Staubli VAL3: io_System.pjx

--- io_System.pjx ---
Parameters version=s7.0 stackSize=5000 millimeterUnit=true
Program file=_globals.pgx
Program file=InitSysIO.pgx
Program file=SysIN.pgx
Program file=SysOUT.pgx
Data file=io_System.dtx
Library alias=io path=Disk://io/io.pjx

--- io_System.dtx ---
public num nLiAuto
public num nLiAux1
public num nLiAux2
public num nLiAux3
public num nLiDoorOpen
public num nLiEnd
public num nLiHome = 1
public num nLiMouldFree
public num nLiPartMade
public num nLiRobotOff
public num nLiSafety
public num nLiStart
public num nLiStop = 1
public num nLiTotalHome = 1
public num nLiWarning
public num nStateRobot
public num nLiTowerRed
public num nLiTowerYellow
public num nLiTowerGreen
public num nPowerCountCtrl
public num nLastServiceCtr
public num nLastServiceArm
public num nServiceRemain
public string sAux1
public string sAux2
public bool bBlockedCycle
public bool bBlockedUser
public bool bBtEnd
public bool bBtHome
public bool bBtRobotOff
public bool bBtStart
public bool bBtStop
public bool bCancelHomeCycl
public bool bCycleEndCalled
public bool bCycleEndPos
public bool bEnd
public bool bF7
public bool bF8
public bool bF_End
public bool bF_Home
public bool bF_Off
public bool bF_Start
public bool bF_Stop
public bool bFirstRunAfterL = true
public bool bFlashFast
public bool bFlashSlow
public bool bForceHomeReq
public bool bForceHome_ = true
public bool bHomeRetActive
public bool bModified
public bool bMouldArmInPLC
public bool bPartMade
public bool bRobotHome = true
public bool bRobotOff
public bool bRobotOffCalled
public bool bRobotOffPos
public bool bRobotZero
public bool bStartHomeCycle
public bool bStartProdCycle
public bool bTotalHome = true
public bool bUsrError
public bool btAux1
public bool btAux2
public bool btAux3
public bool bUsrWarningLow
public bool canStart
public bool canStop
public bool canResume
public bool canHom
public bool canRobotOff
public bool bRecordForce
public bool bErrorAck
public bool bUsrWarningHigh
public bool bIsEmulator
public bool bCancelEndCycle
public bool bStartInEndCycl
public jointRx jEnvMax = {j1=88.269052, j2=85.051261, j3=143.532119, j4=182.33531, j5=117.927529, j6=254.739889}
public jointRx jEnvMin = {j1=-180, j2=-47.382245, j3=-142.046726, j4=-131.97883, j5=-69.877872, j6=-189.153148}
public jointRx jPosErrCurrent = {j1=5.7E-05, j4=6.1E-05}
public jointRx jTorqueCurrent
public aio aiGrip[9]
public dio diArm[9]
public dio diBtAux1
public dio diBtAux2
public dio diBtAux3
public dio diBtEnd
public dio diBtHome
public dio diBtRobotOff
public dio diBtStart
public dio diBtStop
public dio diBtTotalHome
public dio diCore1Pos1
public dio diCore1Pos2
public dio diCore2Pos1
public dio diCore2Pos2
public dio diEjcIn
public dio diEjcOut
public dio diGrip[9]
public dio diGrip2[9]
public dio diLifeBit[2]
public dio diMachineInAuto
public dio diMouldClosed
public dio diMouldFreeFBK
public dio diMouldMidOpen
public dio diMouldOpen
public dio diRejectPart
public dio diSecuFBK[2]
public dio doAir[9]
public dio doArm[9]
public dio doAux1
public dio doAux2
public dio doCore1Pos1
public dio doCore1Pos2
public dio doCore2Pos1
public dio doCore2Pos2
public dio doEjcIn
public dio doEjcOut
public dio doFullOpening
public dio doGrip[9]
public dio doLiAuto
public dio doLiAux1
public dio doLiAux2
public dio doLiAux3
public dio doLiEnd
public dio doLiHome
public dio doLiRobotOff
public dio doLiSafety
public dio doLiStart
public dio doLiStop
public dio doLiTotalHome
public dio doMouldFree
public dio doRobotOff
public dio doSecu[2]
public dio doStartMachine
public dio doLiTowerGreen
public dio doLiTowerYellow
public dio doLiTowerRed
public dio doLiAreaFree
public dio diFuseOK[6]
public dio diSafetyPLC_OK
public dio doSignalHorn
public dio diAC_OK
public dio diLifebitsys = {link=ModbusSrv-0\Plastics-Bit\LifeBitSys}
public dio diUnusedsys = {link=ModbusSrv-0\Plastics-Bit\UnusedSys}
public dio diLifebituser = {link=ModbusSrv-0\Plastics-Bit\LifeBitUser}
public dio diUnuseduser = {link=ModbusSrv-0\Plastics-Bit\UnusedUser}
public dio diSharedbitin[32]
  [0] = {link=ModbusSrv-0\Plastics-Bit\sharedBitIn:32[0]}
  [1] = {link=ModbusSrv-0\Plastics-Bit\sharedBitIn:32[1]}
  [2] = {link=ModbusSrv-0\Plastics-Bit\sharedBitIn:32[2]}
  [3] = {link=ModbusSrv-0\Plastics-Bit\sharedBitIn:32[3]}
  [4] = {link=ModbusSrv-0\Plastics-Bit\sharedBitIn:32[4]}
  [5] = {link=ModbusSrv-0\Plastics-Bit\sharedBitIn:32[5]}
  [6] = {link=ModbusSrv-0\Plastics-Bit\sharedBitIn:32[6]}
  [7] = {link=ModbusSrv-0\Plastics-Bit\sharedBitIn:32[7]}
  [8] = {link=ModbusSrv-0\Plastics-Bit\sharedBitIn:32[8]}
  [9] = {link=ModbusSrv-0\Plastics-Bit\sharedBitIn:32[9]}
  [10] = {link=ModbusSrv-0\Plastics-Bit\sharedBitIn:32[10]}
  [11] = {link=ModbusSrv-0\Plastics-Bit\sharedBitIn:32[11]}
  [12] = {link=ModbusSrv-0\Plastics-Bit\sharedBitIn:32[12]}
  [13] = {link=ModbusSrv-0\Plastics-Bit\sharedBitIn:32[13]}
  [14] = {link=ModbusSrv-0\Plastics-Bit\sharedBitIn:32[14]}
  [15] = {link=ModbusSrv-0\Plastics-Bit\sharedBitIn:32[15]}
  [16] = {link=ModbusSrv-0\Plastics-Bit\sharedBitIn:32[16]}
  [17] = {link=ModbusSrv-0\Plastics-Bit\sharedBitIn:32[17]}
  [18] = {link=ModbusSrv-0\Plastics-Bit\sharedBitIn:32[18]}
  [19] = {link=ModbusSrv-0\Plastics-Bit\sharedBitIn:32[19]}
  [20] = {link=ModbusSrv-0\Plastics-Bit\sharedBitIn:32[20]}
  [21] = {link=ModbusSrv-0\Plastics-Bit\sharedBitIn:32[21]}
  [22] = {link=ModbusSrv-0\Plastics-Bit\sharedBitIn:32[22]}
  [23] = {link=ModbusSrv-0\Plastics-Bit\sharedBitIn:32[23]}
  [24] = {link=ModbusSrv-0\Plastics-Bit\sharedBitIn:32[24]}
  [25] = {link=ModbusSrv-0\Plastics-Bit\sharedBitIn:32[25]}
  [26] = {link=ModbusSrv-0\Plastics-Bit\sharedBitIn:32[26]}
  [27] = {link=ModbusSrv-0\Plastics-Bit\sharedBitIn:32[27]}
  [28] = {link=ModbusSrv-0\Plastics-Bit\sharedBitIn:32[28]}
  [29] = {link=ModbusSrv-0\Plastics-Bit\sharedBitIn:32[29]}
  [30] = {link=ModbusSrv-0\Plastics-Bit\sharedBitIn:32[30]}
  [31] = {link=ModbusSrv-0\Plastics-Bit\sharedBitIn:32[31]}
public dio diReserved1[63]
  [0] = {link=ModbusSrv-0\Plastics-Bit\reserved1:63[0]}
  [1] = {link=ModbusSrv-0\Plastics-Bit\reserved1:63[1]}
  [2] = {link=ModbusSrv-0\Plastics-Bit\reserved1:63[2]}
  [3] = {link=ModbusSrv-0\Plastics-Bit\reserved1:63[3]}
  [4] = {link=ModbusSrv-0\Plastics-Bit\reserved1:63[4]}
  [5] = {link=ModbusSrv-0\Plastics-Bit\reserved1:63[5]}
  [6] = {link=ModbusSrv-0\Plastics-Bit\reserved1:63[6]}
  [7] = {link=ModbusSrv-0\Plastics-Bit\reserved1:63[7]}
  [8] = {link=ModbusSrv-0\Plastics-Bit\reserved1:63[8]}
  [9] = {link=ModbusSrv-0\Plastics-Bit\reserved1:63[9]}
  [10] = {link=ModbusSrv-0\Plastics-Bit\reserved1:63[10]}
  [11] = {link=ModbusSrv-0\Plastics-Bit\reserved1:63[11]}
  [12] = {link=ModbusSrv-0\Plastics-Bit\reserved1:63[12]}
  [13] = {link=ModbusSrv-0\Plastics-Bit\reserved1:63[13]}
  [14] = {link=ModbusSrv-0\Plastics-Bit\reserved1:63[14]}
  [15] = {link=ModbusSrv-0\Plastics-Bit\reserved1:63[15]}
  [16] = {link=ModbusSrv-0\Plastics-Bit\reserved1:63[16]}
  [17] = {link=ModbusSrv-0\Plastics-Bit\reserved1:63[17]}
  [18] = {link=ModbusSrv-0\Plastics-Bit\reserved1:63[18]}
  [19] = {link=ModbusSrv-0\Plastics-Bit\reserved1:63[19]}
  [20] = {link=ModbusSrv-0\Plastics-Bit\reserved1:63[20]}
  [21] = {link=ModbusSrv-0\Plastics-Bit\reserved1:63[21]}
  [22] = {link=ModbusSrv-0\Plastics-Bit\reserved1:63[22]}
  [23] = {link=ModbusSrv-0\Plastics-Bit\reserved1:63[23]}
  [24] = {link=ModbusSrv-0\Plastics-Bit\reserved1:63[24]}
  [25] = {link=ModbusSrv-0\Plastics-Bit\reserved1:63[25]}
  [26] = {link=ModbusSrv-0\Plastics-Bit\reserved1:63[26]}
  [27] = {link=ModbusSrv-0\Plastics-Bit\reserved1:63[27]}
  [28] = {link=ModbusSrv-0\Plastics-Bit\reserved1:63[28]}
  [29] = {link=ModbusSrv-0\Plastics-Bit\reserved1:63[29]}
  [30] = {link=ModbusSrv-0\Plastics-Bit\reserved1:63[30]}
  [31] = {link=ModbusSrv-0\Plastics-Bit\reserved1:63[31]}
  [32] = {link=ModbusSrv-0\Plastics-Bit\reserved1:63[32]}
  [33] = {link=ModbusSrv-0\Plastics-Bit\reserved1:63[33]}
  [34] = {link=ModbusSrv-0\Plastics-Bit\reserved1:63[34]}
  [35] = {link=ModbusSrv-0\Plastics-Bit\reserved1:63[35]}
  [36] = {link=ModbusSrv-0\Plastics-Bit\reserved1:63[36]}
  [37] = {link=ModbusSrv-0\Plastics-Bit\reserved1:63[37]}
  [38] = {link=ModbusSrv-0\Plastics-Bit\reserved1:63[38]}
  [39] = {link=ModbusSrv-0\Plastics-Bit\reserved1:63[39]}
  [40] = {link=ModbusSrv-0\Plastics-Bit\reserved1:63[40]}
  [41] = {link=ModbusSrv-0\Plastics-Bit\reserved1:63[41]}
  [42] = {link=ModbusSrv-0\Plastics-Bit\reserved1:63[42]}
  [43] = {link=ModbusSrv-0\Plastics-Bit\reserved1:63[43]}
  [44] = {link=ModbusSrv-0\Plastics-Bit\reserved1:63[44]}
  [45] = {link=ModbusSrv-0\Plastics-Bit\reserved1:63[45]}
  [46] = {link=ModbusSrv-0\Plastics-Bit\reserved1:63[46]}
  [47] = {link=ModbusSrv-0\Plastics-Bit\reserved1:63[47]}
  [48] = {link=ModbusSrv-0\Plastics-Bit\reserved1:63[48]}
  [49] = {link=ModbusSrv-0\Plastics-Bit\reserved1:63[49]}
  [50] = {link=ModbusSrv-0\Plastics-Bit\reserved1:63[50]}
  [51] = {link=ModbusSrv-0\Plastics-Bit\reserved1:63[51]}
  [52] = {link=ModbusSrv-0\Plastics-Bit\reserved1:63[52]}
  [53] = {link=ModbusSrv-0\Plastics-Bit\reserved1:63[53]}
  [54] = {link=ModbusSrv-0\Plastics-Bit\reserved1:63[54]}
  [55] = {link=ModbusSrv-0\Plastics-Bit\reserved1:63[55]}
  [56] = {link=ModbusSrv-0\Plastics-Bit\reserved1:63[56]}
  [57] = {link=ModbusSrv-0\Plastics-Bit\reserved1:63[57]}
  [58] = {link=ModbusSrv-0\Plastics-Bit\reserved1:63[58]}
  [59] = {link=ModbusSrv-0\Plastics-Bit\reserved1:63[59]}
  [60] = {link=ModbusSrv-0\Plastics-Bit\reserved1:63[60]}
  [61] = {link=ModbusSrv-0\Plastics-Bit\reserved1:63[61]}
  [62] = {link=ModbusSrv-0\Plastics-Bit\reserved1:63[62]}
public dio doN1_102[8]
  [0] = {link=ModbusSrv-0\Plastics-Bit\N1_102:8[0]}
  [1] = {link=ModbusSrv-0\Plastics-Bit\N1_102:8[1]}
  [2] = {link=ModbusSrv-0\Plastics-Bit\N1_102:8[2]}
  [3] = {link=ModbusSrv-0\Plastics-Bit\N1_102:8[3]}
  [4] = {link=ModbusSrv-0\Plastics-Bit\N1_102:8[4]}
  [5] = {link=ModbusSrv-0\Plastics-Bit\N1_102:8[5]}
  [6] = {link=ModbusSrv-0\Plastics-Bit\N1_102:8[6]}
  [7] = {link=ModbusSrv-0\Plastics-Bit\N1_102:8[7]}
public dio doN1_103[8]
  [0] = {link=ModbusSrv-0\Plastics-Bit\N1_103:8[0]}
  [1] = {link=ModbusSrv-0\Plastics-Bit\N1_103:8[1]}
  [2] = {link=ModbusSrv-0\Plastics-Bit\N1_103:8[2]}
  [3] = {link=ModbusSrv-0\Plastics-Bit\N1_103:8[3]}
  [4] = {link=ModbusSrv-0\Plastics-Bit\N1_103:8[4]}
  [5] = {link=ModbusSrv-0\Plastics-Bit\N1_103:8[5]}
  [6] = {link=ModbusSrv-0\Plastics-Bit\N1_103:8[6]}
  [7] = {link=ModbusSrv-0\Plastics-Bit\N1_103:8[7]}
public dio doN1_202[8]
  [0] = {link=ModbusSrv-0\Plastics-Bit\N1_202:8[0]}
  [1] = {link=ModbusSrv-0\Plastics-Bit\N1_202:8[1]}
  [2] = {link=ModbusSrv-0\Plastics-Bit\N1_202:8[2]}
  [3] = {link=ModbusSrv-0\Plastics-Bit\N1_202:8[3]}
  [4] = {link=ModbusSrv-0\Plastics-Bit\N1_202:8[4]}
  [5] = {link=ModbusSrv-0\Plastics-Bit\N1_202:8[5]}
  [6] = {link=ModbusSrv-0\Plastics-Bit\N1_202:8[6]}
  [7] = {link=ModbusSrv-0\Plastics-Bit\N1_202:8[7]}
public dio doN1_303[4]
  [0] = {link=ModbusSrv-0\Plastics-Bit\N1_303:4[0]}
  [1] = {link=ModbusSrv-0\Plastics-Bit\N1_303:4[1]}
  [2] = {link=ModbusSrv-0\Plastics-Bit\N1_303:4[2]}
  [3] = {link=ModbusSrv-0\Plastics-Bit\N1_303:4[3]}
public dio doN1_305[2]
  [0] = {link=ModbusSrv-0\Plastics-Bit\N1_305:2[0]}
  [1] = {link=ModbusSrv-0\Plastics-Bit\N1_305:2[1]}
public dio doN1_306[2]
  [0] = {link=ModbusSrv-0\Plastics-Bit\N1_306:2[0]}
  [1] = {link=ModbusSrv-0\Plastics-Bit\N1_306:2[1]}
public dio doN1_307[2]
  [0] = {link=ModbusSrv-0\Plastics-Bit\N1_307:2[0]}
  [1] = {link=ModbusSrv-0\Plastics-Bit\N1_307:2[1]}
public dio doN1_308[2]
  [0] = {link=ModbusSrv-0\Plastics-Bit\N1_308:2[0]}
  [1] = {link=ModbusSrv-0\Plastics-Bit\N1_308:2[1]}
public dio doN1_309[2]
  [0] = {link=ModbusSrv-0\Plastics-Bit\N1_309:2[0]}
  [1] = {link=ModbusSrv-0\Plastics-Bit\N1_309:2[1]}
public dio doN2_104[8]
  [0] = {link=ModbusSrv-0\Plastics-Bit\N2_104:8[0]}
  [1] = {link=ModbusSrv-0\Plastics-Bit\N2_104:8[1]}
  [2] = {link=ModbusSrv-0\Plastics-Bit\N2_104:8[2]}
  [3] = {link=ModbusSrv-0\Plastics-Bit\N2_104:8[3]}
  [4] = {link=ModbusSrv-0\Plastics-Bit\N2_104:8[4]}
  [5] = {link=ModbusSrv-0\Plastics-Bit\N2_104:8[5]}
  [6] = {link=ModbusSrv-0\Plastics-Bit\N2_104:8[6]}
  [7] = {link=ModbusSrv-0\Plastics-Bit\N2_104:8[7]}
public dio doN2_105[8]
  [0] = {link=ModbusSrv-0\Plastics-Bit\N2_105:8[0]}
  [1] = {link=ModbusSrv-0\Plastics-Bit\N2_105:8[1]}
  [2] = {link=ModbusSrv-0\Plastics-Bit\N2_105:8[2]}
  [3] = {link=ModbusSrv-0\Plastics-Bit\N2_105:8[3]}
  [4] = {link=ModbusSrv-0\Plastics-Bit\N2_105:8[4]}
  [5] = {link=ModbusSrv-0\Plastics-Bit\N2_105:8[5]}
  [6] = {link=ModbusSrv-0\Plastics-Bit\N2_105:8[6]}
  [7] = {link=ModbusSrv-0\Plastics-Bit\N2_105:8[7]}
public dio doN2_106[8]
  [0] = {link=ModbusSrv-0\Plastics-Bit\N2_106:8[0]}
  [1] = {link=ModbusSrv-0\Plastics-Bit\N2_106:8[1]}
  [2] = {link=ModbusSrv-0\Plastics-Bit\N2_106:8[2]}
  [3] = {link=ModbusSrv-0\Plastics-Bit\N2_106:8[3]}
  [4] = {link=ModbusSrv-0\Plastics-Bit\N2_106:8[4]}
  [5] = {link=ModbusSrv-0\Plastics-Bit\N2_106:8[5]}
  [6] = {link=ModbusSrv-0\Plastics-Bit\N2_106:8[6]}
  [7] = {link=ModbusSrv-0\Plastics-Bit\N2_106:8[7]}
public dio doN2_107[8]
  [0] = {link=ModbusSrv-0\Plastics-Bit\N2_107:8[0]}
  [1] = {link=ModbusSrv-0\Plastics-Bit\N2_107:8[1]}
  [2] = {link=ModbusSrv-0\Plastics-Bit\N2_107:8[2]}
  [3] = {link=ModbusSrv-0\Plastics-Bit\N2_107:8[3]}
  [4] = {link=ModbusSrv-0\Plastics-Bit\N2_107:8[4]}
  [5] = {link=ModbusSrv-0\Plastics-Bit\N2_107:8[5]}
  [6] = {link=ModbusSrv-0\Plastics-Bit\N2_107:8[6]}
  [7] = {link=ModbusSrv-0\Plastics-Bit\N2_107:8[7]}
public dio doSharedbitout[32]
  [0] = {link=ModbusSrv-0\Plastics-Bit\sharedBitOut:32[0]}
  [1] = {link=ModbusSrv-0\Plastics-Bit\sharedBitOut:32[1]}
  [2] = {link=ModbusSrv-0\Plastics-Bit\sharedBitOut:32[2]}
  [3] = {link=ModbusSrv-0\Plastics-Bit\sharedBitOut:32[3]}
  [4] = {link=ModbusSrv-0\Plastics-Bit\sharedBitOut:32[4]}
  [5] = {link=ModbusSrv-0\Plastics-Bit\sharedBitOut:32[5]}
  [6] = {link=ModbusSrv-0\Plastics-Bit\sharedBitOut:32[6]}
  [7] = {link=ModbusSrv-0\Plastics-Bit\sharedBitOut:32[7]}
  [8] = {link=ModbusSrv-0\Plastics-Bit\sharedBitOut:32[8]}
  [9] = {link=ModbusSrv-0\Plastics-Bit\sharedBitOut:32[9]}
  [10] = {link=ModbusSrv-0\Plastics-Bit\sharedBitOut:32[10]}
  [11] = {link=ModbusSrv-0\Plastics-Bit\sharedBitOut:32[11]}
  [12] = {link=ModbusSrv-0\Plastics-Bit\sharedBitOut:32[12]}
  [13] = {link=ModbusSrv-0\Plastics-Bit\sharedBitOut:32[13]}
  [14] = {link=ModbusSrv-0\Plastics-Bit\sharedBitOut:32[14]}
  [15] = {link=ModbusSrv-0\Plastics-Bit\sharedBitOut:32[15]}
  [16] = {link=ModbusSrv-0\Plastics-Bit\sharedBitOut:32[16]}
  [17] = {link=ModbusSrv-0\Plastics-Bit\sharedBitOut:32[17]}
  [18] = {link=ModbusSrv-0\Plastics-Bit\sharedBitOut:32[18]}
  [19] = {link=ModbusSrv-0\Plastics-Bit\sharedBitOut:32[19]}
  [20] = {link=ModbusSrv-0\Plastics-Bit\sharedBitOut:32[20]}
  [21] = {link=ModbusSrv-0\Plastics-Bit\sharedBitOut:32[21]}
  [22] = {link=ModbusSrv-0\Plastics-Bit\sharedBitOut:32[22]}
  [23] = {link=ModbusSrv-0\Plastics-Bit\sharedBitOut:32[23]}
  [24] = {link=ModbusSrv-0\Plastics-Bit\sharedBitOut:32[24]}
  [25] = {link=ModbusSrv-0\Plastics-Bit\sharedBitOut:32[25]}
  [26] = {link=ModbusSrv-0\Plastics-Bit\sharedBitOut:32[26]}
  [27] = {link=ModbusSrv-0\Plastics-Bit\sharedBitOut:32[27]}
  [28] = {link=ModbusSrv-0\Plastics-Bit\sharedBitOut:32[28]}
  [29] = {link=ModbusSrv-0\Plastics-Bit\sharedBitOut:32[29]}
  [30] = {link=ModbusSrv-0\Plastics-Bit\sharedBitOut:32[30]}
  [31] = {link=ModbusSrv-0\Plastics-Bit\sharedBitOut:32[31]}
public dio doBrakeselect = {link=ModbusSrv-0\Plastics-Bit\brakeSelect}
public dio doDoor = {link=ModbusSrv-0\Plastics-Bit\door}
public dio doEstopes34 = {link=ModbusSrv-0\Plastics-Bit\estopES34}
public dio doEstopes12 = {link=ModbusSrv-0\Plastics-Bit\estopES12}
public dio doEstopmcp = {link=ModbusSrv-0\Plastics-Bit\estopMCP}
public dio doLimitswitch = {link=ModbusSrv-0\Plastics-Bit\limitSwitch}
public dio doDdummy[8]
  [0] = {link=ModbusSrv-0\Plastics-Bit\dDummy:8[0]}
  [1] = {link=ModbusSrv-0\Plastics-Bit\dDummy:8[1]}
  [2] = {link=ModbusSrv-0\Plastics-Bit\dDummy:8[2]}
  [3] = {link=ModbusSrv-0\Plastics-Bit\dDummy:8[3]}
  [4] = {link=ModbusSrv-0\Plastics-Bit\dDummy:8[4]}
  [5] = {link=ModbusSrv-0\Plastics-Bit\dDummy:8[5]}
  [6] = {link=ModbusSrv-0\Plastics-Bit\dDummy:8[6]}
  [7] = {link=ModbusSrv-0\Plastics-Bit\dDummy:8[7]}
public dio doPower = {link=ModbusSrv-0\Plastics-Bit\power}
public dio doByte0[8]
  [0] = {link=ModbusSrv-0\Plastics-Bit\byte0:8[0]}
  [1] = {link=ModbusSrv-0\Plastics-Bit\byte0:8[1]}
  [2] = {link=ModbusSrv-0\Plastics-Bit\byte0:8[2]}
  [3] = {link=ModbusSrv-0\Plastics-Bit\byte0:8[3]}
  [4] = {link=ModbusSrv-0\Plastics-Bit\byte0:8[4]}
  [5] = {link=ModbusSrv-0\Plastics-Bit\byte0:8[5]}
  [6] = {link=ModbusSrv-0\Plastics-Bit\byte0:8[6]}
  [7] = {link=ModbusSrv-0\Plastics-Bit\byte0:8[7]}
public dio doByte1[8]
  [0] = {link=ModbusSrv-0\Plastics-Bit\byte1:8[0]}
  [1] = {link=ModbusSrv-0\Plastics-Bit\byte1:8[1]}
  [2] = {link=ModbusSrv-0\Plastics-Bit\byte1:8[2]}
  [3] = {link=ModbusSrv-0\Plastics-Bit\byte1:8[3]}
  [4] = {link=ModbusSrv-0\Plastics-Bit\byte1:8[4]}
  [5] = {link=ModbusSrv-0\Plastics-Bit\byte1:8[5]}
  [6] = {link=ModbusSrv-0\Plastics-Bit\byte1:8[6]}
  [7] = {link=ModbusSrv-0\Plastics-Bit\byte1:8[7]}
public dio doByte2[8]
  [0] = {link=ModbusSrv-0\Plastics-Bit\byte2:8[0]}
  [1] = {link=ModbusSrv-0\Plastics-Bit\byte2:8[1]}
  [2] = {link=ModbusSrv-0\Plastics-Bit\byte2:8[2]}
  [3] = {link=ModbusSrv-0\Plastics-Bit\byte2:8[3]}
  [4] = {link=ModbusSrv-0\Plastics-Bit\byte2:8[4]}
  [5] = {link=ModbusSrv-0\Plastics-Bit\byte2:8[5]}
  [6] = {link=ModbusSrv-0\Plastics-Bit\byte2:8[6]}
  [7] = {link=ModbusSrv-0\Plastics-Bit\byte2:8[7]}
public dio doByte3[8]
  [0] = {link=ModbusSrv-0\Plastics-Bit\byte3:8[0]}
  [1] = {link=ModbusSrv-0\Plastics-Bit\byte3:8[1]}
  [2] = {link=ModbusSrv-0\Plastics-Bit\byte3:8[2]}
  [3] = {link=ModbusSrv-0\Plastics-Bit\byte3:8[3]}
  [4] = {link=ModbusSrv-0\Plastics-Bit\byte3:8[4]}
  [5] = {link=ModbusSrv-0\Plastics-Bit\byte3:8[5]}
  [6] = {link=ModbusSrv-0\Plastics-Bit\byte3:8[6]}
  [7] = {link=ModbusSrv-0\Plastics-Bit\byte3:8[7]}
public dio doAgripper[16]
  [0] = {link=ModbusSrv-0\Plastics-Bit\aGripper:16[0]}
  [1] = {link=ModbusSrv-0\Plastics-Bit\aGripper:16[1]}
  [2] = {link=ModbusSrv-0\Plastics-Bit\aGripper:16[2]}
  [3] = {link=ModbusSrv-0\Plastics-Bit\aGripper:16[3]}
  [4] = {link=ModbusSrv-0\Plastics-Bit\aGripper:16[4]}
  [5] = {link=ModbusSrv-0\Plastics-Bit\aGripper:16[5]}
  [6] = {link=ModbusSrv-0\Plastics-Bit\aGripper:16[6]}
  [7] = {link=ModbusSrv-0\Plastics-Bit\aGripper:16[7]}
  [8] = {link=ModbusSrv-0\Plastics-Bit\aGripper:16[8]}
  [9] = {link=ModbusSrv-0\Plastics-Bit\aGripper:16[9]}
  [10] = {link=ModbusSrv-0\Plastics-Bit\aGripper:16[10]}
  [11] = {link=ModbusSrv-0\Plastics-Bit\aGripper:16[11]}
  [12] = {link=ModbusSrv-0\Plastics-Bit\aGripper:16[12]}
  [13] = {link=ModbusSrv-0\Plastics-Bit\aGripper:16[13]}
  [14] = {link=ModbusSrv-0\Plastics-Bit\aGripper:16[14]}
  [15] = {link=ModbusSrv-0\Plastics-Bit\aGripper:16[15]}
public aio aiDummyword[2]
  [0] = {link=ModbusSrv-0\Plastics-Word\dummyWord:2[0]}
  [1] = {link=ModbusSrv-0\Plastics-Word\dummyWord:2[1]}
public aio aiN1_200[4]
  [0] = {link=ModbusSrv-0\Plastics-Word\N1_200:4[0]}
  [1] = {link=ModbusSrv-0\Plastics-Word\N1_200:4[1]}
  [2] = {link=ModbusSrv-0\Plastics-Word\N1_200:4[2]}
  [3] = {link=ModbusSrv-0\Plastics-Word\N1_200:4[3]}
public aio aiSharedwordin[16]
  [0] = {link=ModbusSrv-0\Plastics-Word\sharedWordIn:16[0]}
  [1] = {link=ModbusSrv-0\Plastics-Word\sharedWordIn:16[1]}
  [2] = {link=ModbusSrv-0\Plastics-Word\sharedWordIn:16[2]}
  [3] = {link=ModbusSrv-0\Plastics-Word\sharedWordIn:16[3]}
  [4] = {link=ModbusSrv-0\Plastics-Word\sharedWordIn:16[4]}
  [5] = {link=ModbusSrv-0\Plastics-Word\sharedWordIn:16[5]}
  [6] = {link=ModbusSrv-0\Plastics-Word\sharedWordIn:16[6]}
  [7] = {link=ModbusSrv-0\Plastics-Word\sharedWordIn:16[7]}
  [8] = {link=ModbusSrv-0\Plastics-Word\sharedWordIn:16[8]}
  [9] = {link=ModbusSrv-0\Plastics-Word\sharedWordIn:16[9]}
  [10] = {link=ModbusSrv-0\Plastics-Word\sharedWordIn:16[10]}
  [11] = {link=ModbusSrv-0\Plastics-Word\sharedWordIn:16[11]}
  [12] = {link=ModbusSrv-0\Plastics-Word\sharedWordIn:16[12]}
  [13] = {link=ModbusSrv-0\Plastics-Word\sharedWordIn:16[13]}
  [14] = {link=ModbusSrv-0\Plastics-Word\sharedWordIn:16[14]}
  [15] = {link=ModbusSrv-0\Plastics-Word\sharedWordIn:16[15]}
public aio aiSharedwordout[16]
  [0] = {link=ModbusSrv-0\Plastics-Word\sharedWordOut:16[0]}
  [1] = {link=ModbusSrv-0\Plastics-Word\sharedWordOut:16[1]}
  [2] = {link=ModbusSrv-0\Plastics-Word\sharedWordOut:16[2]}
  [3] = {link=ModbusSrv-0\Plastics-Word\sharedWordOut:16[3]}
  [4] = {link=ModbusSrv-0\Plastics-Word\sharedWordOut:16[4]}
  [5] = {link=ModbusSrv-0\Plastics-Word\sharedWordOut:16[5]}
  [6] = {link=ModbusSrv-0\Plastics-Word\sharedWordOut:16[6]}
  [7] = {link=ModbusSrv-0\Plastics-Word\sharedWordOut:16[7]}
  [8] = {link=ModbusSrv-0\Plastics-Word\sharedWordOut:16[8]}
  [9] = {link=ModbusSrv-0\Plastics-Word\sharedWordOut:16[9]}
  [10] = {link=ModbusSrv-0\Plastics-Word\sharedWordOut:16[10]}
  [11] = {link=ModbusSrv-0\Plastics-Word\sharedWordOut:16[11]}
  [12] = {link=ModbusSrv-0\Plastics-Word\sharedWordOut:16[12]}
  [13] = {link=ModbusSrv-0\Plastics-Word\sharedWordOut:16[13]}
  [14] = {link=ModbusSrv-0\Plastics-Word\sharedWordOut:16[14]}
  [15] = {link=ModbusSrv-0\Plastics-Word\sharedWordOut:16[15]}
public dio N1_100[8] = {link=ModbusSrv-0\Plastics-Bit\N1_100:8[0]}

--- _globals.pgx ---
program _globals()
begin
  //!module
  //\brief
  //This module contains declarations for system IO and system state flags.
  //
  //These variables can be used in a user application.
  //\note
  //This library is typically loaded in a user application using alias <code>SYS:</code>.
  //Therefor, for accessing a member of io_System the SYS: alias identifier has to be prepended, e.g.
  //<code>
  //if SYS:bRobotHome
  //  disablePower()
  //endIf
  //</code>
  //
  //!global nServiceRemain
  //Time given in hours until next service
  //
  //!global nPowerCountCtrl
  //Power count of controller
  //
  //The time the controller has been switched on in h.
  //!global doSignalHorn
  //Digital output to signal horn.
  //
  //The signal horn can be controlled in two ways.\n
  //If setting panel:bSoundOn is true the type of signal indication
  //can be set for each state of the light tower. The settings are available on the MCP display in Advanced -> Edit System Settings ->
  // Sound Indication.\n
  //If setting panel:bSoundOn is false the signal horn is not under the system's control. With this setting the signal horn can be controlled
  //by the user application by controlling signal SYS:doSignalHorn.
  //\sa \ref LightAndSoundIndication
  //\note
  //Output: N1_102[7]; Terminal +XR4.87
  //!global doLiTowerRed
  //Digital output to red light in signal tower.
  //
  //This output is controlled by the system state but it is also controlled by bUsrError.
  //\note
  //Output: N1_103[4]; Terminal +XR4.92
  //\sa nStateRobot, bUsrWarningLow, bUsrWarningHigh, bUsrError, bBlockedUser, \ref LightAndSoundIndication
  //!global doLiTowerYellow
  //Digital output to yellow light in signal tower.
  //
  //This output is controlled by the system state but it is also controlled by bUsrWarningLow and bUsrWarningHigh.
  //\note
  //Output: N1_103[3]; Terminal +XR4.91
  //\sa nStateRobot, bUsrWarningLow, bUsrWarningHigh, bBlockedUser, \ref LightAndSoundIndication
  //!global doLiTowerGreen
  //Digital output to green light in signal tower.
  //
  //This output is on if a robot cycle is active and E-Stop is inactive and bUsrError and bUserWarning are false.
  //\note
  //Output: N1_103[2]; Terminal +XR4.90
  //\sa nStateRobot, bUsrWarningLow, bUsrWarningHigh, bUsrError, \ref LightAndSoundIndication
  //
  //!global bF7
  //\brief
  //is true if the function key F7 on the MCP is pressed.
  //
  //Although the variable has read write access it should only be read by a user program.
  //!global bF8
  //\brief
  //is true if the function key F8 on the MCP is pressed.
  //
  //Although the variable has read write access it should only be read by a user program.
  //!global bF_Start
  //\brief
  //is true if the function key START on the MCP is pressed.
  //
  //Although the variable has read write access it should only be read by a user program.
  //!global bF_Stop
  //\brief
  //is true if the function key STOP on the MCP is pressed.
  //
  //Although the variable has read write access it should only be read by a user program.
  //!global bF_End
  //\brief
  //is true if the function key END on the MCP is pressed.
  //
  //Although the variable has read write access it should only be read by a user program.
  //!global bF_Home
  //\brief
  //is true if the function key HOME on the MCP is pressed.
  //
  //Although the variable has read write access it should only be read by a user program.
  //!global bF_Off
  //\brief
  //is true if the function key ROBOT OFF on the MCP is pressed.
  //
  //Although the variable has read write access it should only be read by a user program.
  //!global bHomeRetActive
  //\brief
  //is true if home return function is running.
  //
  //Although the variable has read write access it should only be read by a user program.
  //!global bPartMade
  //\brief
  //is true if a part has been produced by the machine and the part has not been ejected yet.
  //
  //bPartMade is set to true when the IMM has completely closed the mould.<br>
  //bPartMade is set to false if one of the following conditions is true:
  //<ul>
  //<li>The robot is disabled (ROBOT OFF), the IMM is not in automatic mode and the ejectors have completed a moving sequence.</li>
  //<li>The robot is disabled (ROBOT OFF), the IMM is not in automatic mode and the core 1 has completed a moving sequence.</li>
  //<li>One or more grippers have been closed while the robot is in the mould area.</li>
  //</ul>
  //\note
  //In case of applications where the robot only places parts inside the mould, the variable bPartMade must be explicitly reset in the user program, e.g:
  //<code>
  //movel(pImmPlace, tGripper, mdNormal)
  //waitEndMove()
  ////place insert in mould
  //call FUN:ReleasePart("1")
  ////reset bPartMade to allow next cycle start of IMM
  //SYS:bPartMade=false
  //</code>
  //!global bRobotHome
  //\brief
  //is true if the robot is at its home location.
  //
  //Although the variable has read write access it should only be read by a user program.
  //!global btAux1
  //\brief
  //is true if the key Aux1 is pressed (either on MCP (F7 function key) or on control panel).
  //
  //Although the variable has read write access it should only be read by a user program.
  //!global btAux2
  //\brief
  //is true if the key Aux2 is pressed (either on MCP (F8 function key) or on control panel).
  //
  //Although the variable has read write access it should only be read by a user program.
  //!global btAux3
  //\brief
  //is true if the key Aux3 is pressed (either on MCP or on control panel).
  //
  //Although the variable has read write access it should only be read by a user program.
  //!global aiGrip
  //\brief
  //Analogue gripper feedback signals are linked to this aio array.
  //
  //!global bGrip
  //\brief
  //is an array that represents the state of the gripper feedback signal.
  //
  // If it is true the corresponding gripper has a part gripped.
  //\obsolete
  //!global bModified
  //\brief
  //Indicates if data in the user application have been changed in the "Adjust" menu, e.g. locations
  //
  //!global bMouldFree
  //\brief
  //is true if the flange and the tcp tGripCenter are out of mould area.
  //
  //Although the variable has read write access it should only be read by a user program.
  //!global bRobotZero
  //\brief
  //is true if the robot is at its zero position.
  //
  //Although the variable has read write access it should only be read by a user program.
  //!global bRobotHome
  //\brief
  //is true if the robot is at the home position defined in the currently loaded user application.
  //
  //Although the variable has read write access it should only be read by a user program.
  //!global sAux1
  //\brief
  //A string containing the text that is displayed above the F7 function key.
  //
  //The text is limited to four characters.
  //!global sAux2
  //\brief
  //A string containing the text that is displayed above the F8 function key.
  //
  //The text is limited to four characters.
  //!global bBtStop
  //\brief
  // bBtStop is true if the STOP button is being pressed.
  //
  // The source for the STOP function can be the control bar on the MCP or the digital input.
  //Although the variable has read write access it should only be read by a user program.
  //!global bBtStart
  //\brief
  // bBtStart is true if the START button is being pressed.
  //
  // The source for the START function can be the control bar on the MCP or the digital input.
  //Although the variable has read write access it should only be read by a user program.
  //!global bBtEnd
  //\brief
  // bBtEnd is true if the END button is being pressed.
  //
  // The source for the END function can be the control bar on the MCP or the digital input.
  //Although the variable has read write access it should only be read by a user program.
  //!global bBtHome
  //\brief
  // bBtHome is true if the HOME button is being pressed.
  //
  // The source for the HOME function can be the control bar on the MCP or the digital input.
  //Although the variable has read write access it should only be read by a user program.
  //!global bBtRobotOff
  //\brief
  // bBtRobotOff is true if the ROBOT OFF button is being pressed.
  //
  // The source for the ROBOT OFF function can be the control bar on the MCP or the digital input.
  //Although the variable has read write access it should only be read by a user program.
  //!global bBlockedCycle
  //\brief
  //bBlockedCycle is true if the robot is not moving for the time specified in data:nRobotBlocked
  //during production.
  //
  //This can be due to a signal condition that is missing in the task MP_MainProgram. Check the state
  //of task MP_MainProgram in the task manager.
  //!global bBlockedUser
  //\brief
  //bBlockedUser is true if robot movement is halted by the operator during running production.
  //
  //The robot can be halted by the operator if he presses the Move/Hold button on the MCP and thus
  //puts the robot into hold mode. This condition is also indicated to the operator by a red light
  //on the optionally connected light tower.
  //\sa doLiTowerRed
  //!global bCancelHomeCycl
  //\internal
  //!global bCycleEndCalled
  //\brief
  //is true if the operator has requested a cycle end by pressing the CYCLE END button.
  //
  //bCycleEndCalled is true as long as the robot is busy completing the last cycle or
  //if the operator presses CYCLE END again in order to cancel his previous cycle end request.
  //!global bCancelEndCycle
  //indicates if the operator is allowed to reset a pending "end cycle" request.
  //
  //By default the operator is allowed to reset a "end cycle" request at any time while to robot is active.
  //For some applications it is necessary that a requested "end cycle" function cannot be reset by the
  //operator again. In this case bCancelEndCycle must be set to true.
  //\note
  //Flag bCancelEndCycle is set to true on every cycle start automatically. In order to disallow
  // the function the flag needs to be set to false in the user program, e.g. in the start up section
  //of MP_MainProgram().
  //!global bStartInEndCycl
  //indicates if the IMM is started by calling FUN:StartMachine() in an active "end cycle" request.
  //
  //By default the function FUN:StartMachine() does not start an IMM cycle if the operator has requested
  // an "end cycle". In some applications, however it might be necessary to start an IMM cycle even during
  // a pending "end cycle" request, e.g. in applications where the robot places inserts in the mould and the
  // last cycle includes an IMM cycle with these inserts.
  //\note
  //Flag bStartInEndCycl is set to false on every cycle start automatically. In order to allow
  // the function the flag needs to be set to true in the user program, e.g. in the start up section
  //of MP_MainProgram().
  //!global nStateRobot
  //\brief
  //The value of \a nStateRobot indicates the state of the robot
  //<table>
  //<tr><td>Value</td><td>Description</td></tr>
  //<tr><td>0</td><td>The robot is idling</td></tr>
  //<tr><td>10</td><td>The robot is active and the cycle is running.</td></tr>
  //<tr><td>20</td><td>The robot movement is suspended, production cycle is halted due to a deteced gripper error or the operator has pressed
  //the STOP button, the CYCLE END button or the ROBOT OFF button.</td></tr>
  //<tr><td>25</td><td>The operator has pressed the HOME button while the robot was active (\a nStateRobot==10). The robot movement is suspended, production cycle is halted.</td></tr>
  //<tr><td>32</td><td>The home return function is active.</td></tr>
  //</table>
  //!global bUsrWarningLow
  //is true if an user application has detected a warning condition with low priority.
  //
  //If an user application detects a warning condition (e.g. a feeder is running low with parts), it can inform the operator
  //by setting the variable bUsrWarningLow to true.
  //bUsrWarningLow can be set explicitly by a user application, e.g.:
  //<code>
  //if bAlmostEmpty==true
  //  SYS:bUsrWarningLow=true
  //endIf
  //</code>
  //
  //As a consequence the yellow light on an optionally connected light tower is activated, but the robot cycle continues.
  //bUsrWarningLow must be reset by the user application, e.g.
  //in the home return function HR_HomeReturn().
  //\sa bUsrError, doLiTowerYellow, bUsrWarningHigh
  //!global bUsrWarningHigh
  //is true if an user application has detected a warning condition with high priority.
  //
  //If an user application detects a warning condition that requires immediate attention by the operator
  //(e.g. a feeder is running out of parts), it can inform the operator
  //by setting the variable bUsrWarningHigh to true.
  //bUsrWarningHigh can be set explicitly by a user application, e.g.:
  //<code>
  //if bIsEmpty==true
  //  SYS:bUsrWarningHigh=true
  //endIf
  //</code>
  //
  //As a consequence the yellow light on an optionally connected light tower starts flashing, but the robot cycle continues.
  //bUsrWarningHigh must be reset by the user application, e.g.
  //in the home return function HR_HomeReturn().
  //\sa bUsrError, doLiTowerYellow, bUsrWarningLow
  //!global bUsrError
  //is true if an user application has detected an error condition.
  //
  //If an user application detects an error condition (e.g. a time out in a feeding station, wrongly positioned parts), it can inform the operator
  //by setting the variable bUsrError to true.
  //bUsrError can be set explicitly by a user application, e.g.:
  //<code>
  //if bWrongPart==true
  //  SYS:bUsrError=true
  //endIf
  //</code>
  //bUsrError is implicitly set to true when function FUN:stopMove(string) is being called, e.g.:
  //<code>
  //if bWrongPart==true
  //  call FUN:stopMove("Wrong part in station")
  //endIf
  //</code>
  //
  //As a consequence the red light on an optionally connected light tower is activated and robot motion is being halted.
  //bUsrError is reset to false only if the robot cycle was active and the cycle has been resumed by the operator by pressing START.\n
  //If the operator breaks the cycle by executing a home return, bUsrError does not reset automatically. Thus bUsrError must be reset by the user application, e.g.
  //in the home return function HR_HomeReturn().
  //\sa FUN:stopMove(), bUsrWarningLow, bUsrWarningHigh, doLiTowerRed
  //!global bRecordForce
  //if true force recording in calls to FUN:movelLimited() is active.
  //
  //
  //\page LightAndSoundIndication  Light and Sound Indication
  //
  //The Plastics Innovation software is prepared to control a sound and light indication tower.
  //Below a table of states and their respective light indication:<br>
  //\n
  //Green Light:
  //<table>
  //<tr><td>On</td><td>Robot cycle is active (SYS:nStateRobot = 10)</td></tr>
  //<tr><td>Flashing</td><td>Not defined</td></tr>
  //<tr><td>Off</td><td>Robot cycle is stopped<br>Robot is off / IMM operation without robot</td></tr>
  //</table>
  //\n
  //Yellow Light:
  //<table>
  //<tr><td>On</td><td>Attention needed, low priority (SYS:bUsrWarningLow = true)</td></tr>
  //<tr><td>Flashing</td><td>Attention needed, high priority (SYS:bUsrWarningHigh = true)</td></tr>
  //<tr><td>Off</td><td>Robot is off / IMM operation without robot</td></tr>
  //</table>
  //\n
  //Red Light:
  //<table>
  //<tr><td>On</td><td>Acknowledged alarm pending</td></tr>
  //<tr><td>Flashing</td><td>Alarm pending which is not acknowledged yet by operator</td></tr>
  //<tr><td>Off</td><td>No Alarm pending</td></tr>
  //</table>
  //\n
  //An Alarm is asserted if one of the following conditions has occurred:
  //\li Emergency stop activated
  //\li Gripper fault detected
  //\li Robot cycle blocked (e.g. waiting for signal condition)
  //\li Robot movement suspended by operator (Move/Hold function on MCP)
  //\li User error (bUsrError = true)
end

--- SysIN.pgx ---
program SysIN()
// Initialize system inputs.
  local num idx
begin
  //
  // WAGO Life Bit INPUTS ===============================
  dioLink(diLifeBit[0],io:LifeBitSys)
  dioLink(diLifeBit[1],io:LifeBitUser)
  //
  // ROBOT CONTROL INPUTS (BOTTOMS) =================
  dioLink(diBtStart,io:N1_100[0])
  dioLink(diBtStop,io:N1_100[1])
  dioLink(diBtEnd,io:N1_100[2])
  dioLink(diBtRobotOff,io:N1_100[4])
  dioLink(diBtHome,io:N1_100[3])
  dioLink(diBtTotalHome,io:N1_101[1])
  // AUX FUNTIONS =================================
  dioLink(diBtAux1,io:N1_101[5])
  dioLink(diBtAux2,io:N1_101[6])
  dioLink(diBtAux3,io:N1_101[7])
  // FUSE MONITOR INPUTS ===========================
  for idx=0 to 5
    dioLink(diFuseOK[idx],io:N1_104[idx])
  endFor
//  dioLink(diEM67FuseErr,io:N1_304[1])
//  dioLink(diEM6724VOK,io:N1_304[0])
  // A/C MONITOR INPUTS
  dioLink(diAC_OK,io:N1_104[7])
  // SAFETY PLC MONITOR INPUTS
  dioLink(diSafetyPLC_OK,io:N1_104[7])
  //
  // SAFETY INPUTS ==================================
  dioLink(diMouldFreeFBK,io:N1_302[0])
  dioLink(diSecuFBK[0],io:N1_302[2])
  dioLink(diSecuFBK[1],io:N1_302[3])
  //
  // EUROMAP INPUTS =================================
  dioLink(diRejectPart,io:N1_300[0])
  dioLink(diMouldClosed,io:N1_300[1])
  //  dioLink(diMouldOpen,io:N1_100[5])
  //  dioLink(diMouldMidOpen,io:N1_100[6])
  dioLink(diMouldOpen,io:N1_300[2])
  dioLink(diMouldMidOpen,io:N1_300[3])
  dioLink(diMachineInAuto,io:N1_300[4])
  dioLink(diEjcIn,io:N1_300[5])
  dioLink(diEjcOut,io:N1_300[6])
  dioLink(diCore1Pos1,io:N1_300[7])
  dioLink(diCore1Pos2,io:N1_301[0])
  dioLink(diCore2Pos1,io:N1_301[1])
  dioLink(diCore2Pos2,io:N1_301[2])
  //
end
